// TwinCAT 3 PLC project TimeProjectPLC
// ProgramVersion: 3.1.4024.0
// libraries:
//   EventBufferLibrary, * (Kril GmbH)
//   Tc2_Standard, * (Beckhoff Automation GmbH)
//   Tc2_System, * (Beckhoff Automation GmbH)
//   Tc2_Utilities, * (Beckhoff Automation GmbH)
//   Tc3_Module, * (Beckhoff Automation GmbH)
//   TcUnit, * (www.tcunit.org)
// project tree:
//   / PlcTask.TcTTO
//   POUs/ MAIN.TcPOU
// real-time tasks:
//   TASK PlcTask: cycle T#10ms, priority 20, ADS port 350

CONFIGURATION TimeProjectPLC
    RESOURCE PLC ON TwinCAT3
        TASK PlcTask(INTERVAL := T#10ms, PRIORITY := 20);
        PROGRAM MAIN WITH PlcTask : MAIN;
    END_RESOURCE
END_CONFIGURATION

// ---- POUs/MAIN.TcPOU
PROGRAM MAIN
VAR
	//stThisIsOurFirstInstance : ST_Event;
	bBoolean : BOOL := FALSE;
	
	// Event 1 
	eEventType1 : E_EventType := E_EventType.Alarm;
	eEventSeverity1 : TcEventSeverity := TcEventSeverity.Error;
	nEveventIndentity1: UDINT := 42;
	sEventText1 : STRING(255) := 'This is scary Event 1';
	
		// Event 2 
	eEventType2 : E_EventType := E_EventType.Alarm;
	eEventSeverity2 : TcEventSeverity := TcEventSeverity.Error;
	nEveventIndentity2: UDINT := 43;
	sEventText2 : STRING(255) := 'This is scary Event 2';
	
		// Event 3 
	eEventType3 : E_EventType := E_EventType.Alarm;
	eEventSeverity3 : TcEventSeverity := TcEventSeverity.Error;
	nEveventIndentity3: UDINT := 44;
	sEventText3 : STRING(255) := 'This is scary Eventb 3';
	
	BufferArray : ARRAY [0..(nMAXIMUM_NUMBER_OF_EVENTS *(SIZEOF(ST_Event) +nMEMORY_RING_BUFFER_INTERNAL_EXTRA_SPACING))] OF BYTE;
	fbEventBuffer : FB_EventBuffer(ADR(BufferArray),SIZEOF(BufferArray));
	CsvPersistanceEventStorage : FB_CsvPersistenceEventStorange(fbEventBuffer);
	EventLogger : EventLogger(CsvPersistanceEventStorage);
END_VAR
VAR CONSTANT
	nMAXIMUM_NUMBER_OF_EVENTS : UDINT := 10;
	nMEMORY_RING_BUFFER_INTERNAL_EXTRA_SPACING : INT :=8;
END_VAR



IF bBoolean THEN
	EventLogger.AddEvent(eEventType1, eEventSeverity1, nEveventIndentity1, sEventText1);
	EventLogger.AddEvent(eEventType2, eEventSeverity2, nEveventIndentity2, sEventText2);
	EventLogger.AddEvent(eEventType3, eEventSeverity3, nEveventIndentity3, sEventText3);

	bBoolean := FALSE;
END_IF

CsvPersistanceEventStorage ();

END_PROGRAM
